PROGRAM MAIN
VAR
END_VAR

END_PROGRAM

(* stored: Version 1.1.0.1, ProductVersion 3.1.0.26
   POU MAIN: Id {3a74fcbd-c08b-4030-9a9d-d7e44ec093a7} *)
